(* PLC project Unnamed, Nieznany Unnamed 1 *)
(* stored: creationDateTime 2024-02-24T19:07:32, modificationDateTime 2024-02-24T19:11:07 *)

PROGRAM Nowy
  VAR
    X : DINT;
    Y : DINT;
    Z : DINT;
  END_VAR

STEP S0:
END_STEP
TRANSITION FROM S0 TO (S1, S2)
  := not X;
END_TRANSITION
STEP S1:
END_STEP
TRANSITION FROM (S1, S2) TO S0
  := not (X and Y);
END_TRANSITION
STEP S2:
END_STEP
END_PROGRAM

CONFIGURATION Config0
  RESOURCE Res0 ON PLC
    TASK task0(INTERVAL := T#20ms, PRIORITY := 0);
    PROGRAM instance0 WITH task0 : Nowy;
  END_RESOURCE
END_CONFIGURATION
